// TIA Portal V15 export
// export: Created 2018-05-29T12:25:38.1552518Z, ExportSetting WithDefaults, DisplayName Totally Integrated Automation Portal, DisplayVersion V15, DisplayName STEP 7 Professional, DisplayVersion V15, DisplayName WinCC Professional, DisplayVersion V15, DisplayName TIA Portal Openness, DisplayVersion V15
FUNCTION_BLOCK "phase_example"   // FB1, STL
TITLE = phase_example_fc
{ S7_Optimized_Access := 'TRUE' }
VERSION : 0.1
// phase_example
// This some general description in a comment table.
// This is a new line in the description.
// This is another comment table without borders.
// This is a new line in the 2nd table
// stored: AutoNumber true, UDAEnableTagReadback false
   VAR_INPUT
      scantime : Real;   // the scantime of this EM/phase, used to increase timers
      Bool1 : BOOL;   // - undefined
      Bool2 : BOOL;   // - undefined
      EM_I_OUT_ID : INT;   // - undefined
      Some_Dyn_EM_ID : INT;   // - undefined
      DB_NO : INT;   // - undefined
      XV003_OPN : BOOL;   // - undefined
      XV003_CLS : BOOL;   // - undefined
      XV003_MERR : BOOL;   // - undefined
      XV004_OPN : BOOL;   // - undefined
      XV004_CLS : BOOL;   // - undefined
      XV004_MERR : BOOL;   // - undefined
      XV005_OPN : BOOL;   // - undefined
      XV005_CLS : BOOL;   // - undefined
      XV005_MERR : BOOL;   // - undefined
      P001_RUN : BOOL;   // test a CM - undefined
      P001_STOP : BOOL;   // test a CM - undefined
      P001_MERR : BOOL;   // test a CM - undefined
      P001_MPS : BOOL;   // test a CM - Motor Protecting Switch
      P002_RUN : BOOL;   // test a CM where the casing doesn't match an existing type - undefined
      P002_STOP : BOOL;   // test a CM where the casing doesn't match an existing type - undefined
      P002_MERR : BOOL;   // test a CM where the casing doesn't match an existing type - undefined
      P002_MPS : BOOL;   // test a CM where the casing doesn't match an existing type - Motor Protecting Switch
      EM_I_OUT_OWN : INT;   // - undefined
      EM_I_OUT_STA : INT;   // - undefined
      EM_I_OUT_ERR : BOOL;   // - undefined
      EM_I_OUT_ERRNO : DINT;   // - undefined
      EM_I_OUT_ACTIV : BOOL;   // - undefined
      EM_I_OUT_LT : REAL;   // - undefined
      EM_I_OUT_PT : REAL;   // - undefined
      LT001_PV : REAL;   // - undefined
      LT001_AHH : BOOL;   // - undefined
      LT001_AH : BOOL;   // - undefined
      LT001_AL : BOOL;   // - undefined
      LT001_ALL : BOOL;   // - undefined
      LT001_ERR : BOOL;   // - undefined
      LT002_PV : REAL;   // - undefined
      LT002_AHH : BOOL;   // - undefined
      LT002_AH : BOOL;   // - undefined
      LT002_AL : BOOL;   // - undefined
      LT002_ALL : BOOL;   // - undefined
      LT002_ERR : BOOL;   // - undefined
      FIC001_PV : REAL;   // - undefined
      FIC001_ERR : BOOL;   // - undefined
      Some_Dyn_EM_OWN : INT;   // An example of an EM that's dynamically linked to the phase - undefined
      Some_Dyn_EM_STA : INT;   // An example of an EM that's dynamically linked to the phase - undefined
      Some_Dyn_EM_ERR : BOOL;   // An example of an EM that's dynamically linked to the phase - undefined
      Some_Dyn_EM_ERRNO : DINT;   // An example of an EM that's dynamically linked to the phase - undefined
      Some_Dyn_EM_ACTIV : BOOL;   // An example of an EM that's dynamically linked to the phase - undefined
      Some_Dyn_EM_LT : REAL;   // An example of an EM that's dynamically linked to the phase - undefined
      Some_Dyn_EM_PT : REAL;   // An example of an EM that's dynamically linked to the phase - undefined
      XV008_OPN : BOOL;   // - undefined
      XV008_CLS : BOOL;   // - undefined
      XV008_MERR : BOOL;   // - undefined
   END_VAR
   VAR_OUTPUT
      phase_id : Int;   // unique number for every phase instance over the whole project
      state : Int;
      stepnumber : Int;   // actual stepnumber
      message : DInt;   // number of the message to be displayed
      button_1_text : DInt;   // number of the text to be displayed on the button_1_text
      button_2_text : DInt;   // number of the text to be displayed on the button_2_text
      button_3_text : DInt;   // number of the text to be displayed on the button_3_text
      button_1_visible : Bool;   // 1 = visible
      button_2_visible : Bool;   // 1 = visible
      button_3_visible : Bool;   // 1 = visible
      button_reverse : Byte;   // spare
      state_idle : Bool;
      state_running : Bool;
      state_complete : Bool;
      state_pausing : Bool;
      state_paused : Bool;
      state_holding : Bool;
      state_held : Bool;
      state_restarting : Bool;
      state_stopping : Bool;
      state_stopped : Bool;
      state_aborting : Bool;
      state_aborted : Bool;
      enable_start : Bool;   // 1 start command from hmi or other operator interface
      enable_stop : Bool;   // 2 stop command from hmi or other operator interface
      enable_hold : Bool;   // 3 hold command from hmi or other operator interface
      enable_restart : Bool;   // 4 restart command from hmi or other operator interface
      enable_abort : Bool;   // 5 abort command from hmi or other operator interface
      enable_reset : Bool;   // 6 reset command from hmi or other operator interface
      enable_pause : Bool;   // 7 pause command from hmi or other operator interface
      enable_resume : Bool;   // 8 resume command from hmi or other operator interface
      enable_auto : Bool;   // 1 = auto command from plc program
      enable_man : Bool;   // 1 = manual command from plc program
      enable_byte : Bool;
      auto : Bool;
      steptime_s : Real;   // complete steptime in seconds. same value as the other steptimes
      steptime_m : Real;   // complete steptime in minutes. same value as the other steptimes
      steptime_h : Real;   // complete steptime in hours. same value as the other steptimes
      MSG_no01 : Dint;
      MSG_no02 : Dint;
      MSG_no03 : Dint;
      MSG_no04 : Dint;
      MSG_no05 : Dint;
      MSG_no06 : Dint;
      MSG_no07 : Dint;
      MSG_no08 : Dint;
      MSG_no09 : Dint;
      MSG_no10 : Dint;
      Destination : INT;   // - undefined
      setpoint : REAL;   // - undefined
      some_bool_out : BOOL;   // - undefined
      XV003_CMD : BOOL;   // - Auto command from program
      XV004_CMD : BOOL;   // - Auto command from program
      XV005_CMD : BOOL;   // - Auto command from program
      P001_ON : BOOL;   // test a CM - Switch Motor ON
      P001_AUT : BOOL;   // test a CM - Swtich Motor to AUTO
      P002_ON : BOOL;   // test a CM where the casing doesn't match an existing type - Switch Motor ON
      P002_AUT : BOOL;   // test a CM where the casing doesn't match an existing type - Swtich Motor to AUTO
      EM_I_OUT_REQ : INT;   // - undefined
      EM_I_OUT_CMD : INT;   // - undefined
      EM_I_OUT_P_SP : REAL;   // - undefined
      FIC001_EXT : BOOL;   // - Switch to External Mode
      FIC001_SP : REAL;   // - Operator Setpoint in Internal Mode
      FIC001_AUT : BOOL;   // - Switch to Auto Mode
      FIC001_VAL_OUT : REAL;   // - Operator Output Value
      FIC001_SET_SP : BOOL;   // - undefined
      FIC001_SET_OUT : BOOL;   // - undefined
      Some_Dyn_EM_REQ : INT;   // An example of an EM that's dynamically linked to the phase - undefined
      Some_Dyn_EM_CMD : INT;   // An example of an EM that's dynamically linked to the phase - undefined
      Some_Dyn_EM_P_SP : REAL;   // An example of an EM that's dynamically linked to the phase - undefined
      timer_dosing_pause : BOOL;   // timer paused - undefined
      timer_dosing_s : REAL;   // timer in seconds - undefined
      timer_dosing_m : REAL;   // timer in minutes - undefined
      timer_dosing_h : REAL;   // timer in hours - undefined
      timer_mixing_pause : BOOL;   // timer paused - undefined
      timer_mixing_s : REAL;   // timer in seconds - undefined
      timer_mixing_m : REAL;   // timer in minutes - undefined
      timer_mixing_h : REAL;   // timer in hours - undefined
      timer_circulation_pause : BOOL;   // timer paused - undefined
      timer_circulation_s : REAL;   // timer in seconds - undefined
      timer_circulation_m : REAL;   // timer in minutes - undefined
      timer_circulation_h : REAL;   // timer in hours - undefined
      XV008_CMD : BOOL;   // - Auto command from program
   END_VAR
   VAR_IN_OUT
      plc_commands : DWord;   // combined commands from the master
      hmi_commands : DWord;   // combined commands from the HMI
      hmi_par_without_unit : Real;   // - undefined
      timesetting : Real;   // - undefined
   END_VAR
   VAR DB_SPECIFIC
      previous_stepnumber : Int;   // actual stepnumber
      start_conditions : Bool;   // start conditions 1 = all good
      hold_conditions : Bool;   // hold conditions 1 = all good
      first_scan : Bool;   // first scan of the step active
      last_scan : Bool;   // last scan of the step active
      start_cond_01 : Bool;   // 1 = OK / 0 = NOK
      start_cond_02 : Bool;   // 1 = OK / 0 = NOK
      start_cond_03 : Bool;   // 1 = OK / 0 = NOK
      start_cond_04 : Bool;   // 1 = OK / 0 = NOK
      start_cond_05 : Bool;   // 1 = OK / 0 = NOK
      start_cond_06 : Bool;   // 1 = OK / 0 = NOK
      start_cond_07 : Bool;   // 1 = OK / 0 = NOK
      start_cond_08 : Bool;   // 1 = OK / 0 = NOK
      start_cond_09 : Bool;   // 1 = OK / 0 = NOK
      start_cond_10 : Bool;   // 1 = OK / 0 = NOK
      start_cond_11 : Bool;   // 1 = OK / 0 = NOK
      start_cond_12 : Bool;   // 1 = OK / 0 = NOK
      start_cond_13 : Bool;   // 1 = OK / 0 = NOK
      start_cond_14 : Bool;   // 1 = OK / 0 = NOK
      start_cond_15 : Bool;   // 1 = OK / 0 = NOK
      start_cond_16 : Bool;   // 1 = OK / 0 = NOK
      hold_cond_01 : Bool;   // 1 = OK / 0 = NOK
      hold_cond_02 : Bool;   // 1 = OK / 0 = NOK
      hold_cond_03 : Bool;   // 1 = OK / 0 = NOK
      hold_cond_04 : Bool;   // 1 = OK / 0 = NOK
      hold_cond_05 : Bool;   // 1 = OK / 0 = NOK
      hold_cond_06 : Bool;   // 1 = OK / 0 = NOK
      hold_cond_07 : Bool;   // 1 = OK / 0 = NOK
      hold_cond_08 : Bool;   // 1 = OK / 0 = NOK
      hold_cond_09 : Bool;   // 1 = OK / 0 = NOK
      hold_cond_10 : Bool;   // 1 = OK / 0 = NOK
      hold_cond_11 : Bool;   // 1 = OK / 0 = NOK
      hold_cond_12 : Bool;   // 1 = OK / 0 = NOK
      hold_cond_13 : Bool;   // 1 = OK / 0 = NOK
      hold_cond_14 : Bool;   // 1 = OK / 0 = NOK
      hold_cond_15 : Bool;   // 1 = OK / 0 = NOK
      hold_cond_16 : Bool;   // 1 = OK / 0 = NOK
      in_steprange : Bool;   // detection of steprange for holdcondition
      Module_Error : Bool;   // Error on one of the connected modules (CM or EM)
      CM_Error_no : Dint;   // Error no of the CM in error
      EM_Error_no : Dint;   // Error no of the EM in error
      "e" : Real;   // - undefined
      f : Real;   // - undefined
      g : Real;   // - undefined
      h : Real;   // - undefined
      ii : Real;   // - undefined
      j : Real;   // - undefined
      k : Real;   // - undefined
      l : Real;   // - undefined
      mm : Real;   // - undefined
      n : Real;   // - undefined
      o : Real;   // - undefined
      pp : Real;   // - undefined
      qq : Real;   // - undefined
      rr : Real;   // - undefined
      ss : Real;   // - undefined
      tt : Real;   // - undefined
      u : Real;   // - undefined
      v : Real;   // - undefined
      ww : Real;   // - undefined
      xx : Real;   // - undefined
      y : Real;   // - undefined
      z : Real;   // - undefined
      foo : Real;   // - undefined
      bar : Real;   // - undefined
      stoplevel : Real;   // - undefined
      startlevel : Real;   // - undefined
      offset : Real;   // - undefined
      var1 : Real;   // - undefined
      test1 : Real;   // - undefined
      test2 : Real;   // - undefined
      intvar : Int;   // - undefined
      ""EM_I_OUT"" : "EM_I_OUT_UDT";   // UDT for the linked EM
      ""Some_Dyn_EM"" : "EM_I_OUT_UDT";   // UDT for the linked EM
   END_VAR
   VAR_TEMP
      plc_start : Bool;   // 1 start command from plc program
      plc_stop : Bool;   // 2 stop command from plc program
      plc_hold : Bool;   // 3 hold command from plc program
      plc_restart : Bool;   // 4 restart command from plc program
      plc_abort : Bool;   // 5 abort command from plc program
      plc_reset : Bool;   // 6 reset command from plc program
      plc_pause : Bool;   // 7 pause command from plc program
      plc_resume : Bool;   // 8 resume command from plc program
      plc_auto : Bool;   // 0 manual,1 auto command from plc program
      plc_man : Bool;   // 0 manual,1 auto command from plc program
      plc_cmd : Bool;
      hmi_start : Bool;   // 1 start command from hmi or other operator interface
      hmi_stop : Bool;   // 2 stop command from hmi or other operator interface
      hmi_hold : Bool;   // 3 hold command from hmi or other operator interface
      hmi_restart : Bool;   // 4 restart command from hmi or other operator interface
      hmi_abort : Bool;   // 5 abort command from hmi or other operator interface
      hmi_reset : Bool;   // 6 reset command from hmi or other operator interface
      hmi_pause : Bool;   // 7 pause command from hmi or other operator interface
      hmi_resume : Bool;   // 8 resume command from hmi or other operator interface
      hmi_auto : Bool;   // 1 auto command from plc program
      hmi_man : Bool;   // 0 manual command from plc program
      hmi_cmd : Bool;
      hmi_BTN1 : Bool;
      hmi_BTN2 : Bool;
      hmi_BTN3 : Bool;
      command_start : Bool;   // 1 start command from plc or hmi
      command_stop : Bool;   // 2 stop command from plc or hmi
      command_hold : Bool;   // 3 hold command from plc or hmi
      command_restart : Bool;   // 4 restart command from plc or hmi
      command_abort : Bool;   // 5 abort command from plc or hmi
      command_reset : Bool;   // 6 reset command from plc or hmi
      command_pause : Bool;   // 7 pause command from plc or hmi
      command_resume : Bool;   // 8 resume command from plc or hmi
      command_auto : Bool;   // 1 auto command from plc or hmi
      command_man : Bool;   // 0 auto command from plc or hmi
      command_cmd : Bool;
      button_1_pushed : Bool;   // button pushed
      button_2_pushed : Bool;   // button pushed
      button_3_pushed : Bool;   // button pushed
      sh_cond_01 : Bool;   // 1 = OK / 0 = NOK: intermediate value
      sh_cond_02 : Bool;   // 1 = OK / 0 = NOK: intermediate value
      sh_cond_03 : Bool;   // 1 = OK / 0 = NOK: intermediate value
      sh_cond_04 : Bool;   // 1 = OK / 0 = NOK: intermediate value
      sh_cond_05 : Bool;   // 1 = OK / 0 = NOK: intermediate value
      sh_cond_06 : Bool;   // 1 = OK / 0 = NOK: intermediate value
      sh_cond_07 : Bool;   // 1 = OK / 0 = NOK: intermediate value
      sh_cond_08 : Bool;   // 1 = OK / 0 = NOK: intermediate value
      sh_cond_09 : Bool;   // 1 = OK / 0 = NOK: intermediate value
      sh_cond_10 : Bool;   // 1 = OK / 0 = NOK: intermediate value
      sh_cond_11 : Bool;   // 1 = OK / 0 = NOK: intermediate value
      sh_cond_12 : Bool;   // 1 = OK / 0 = NOK: intermediate value
      sh_cond_13 : Bool;   // 1 = OK / 0 = NOK: intermediate value
      sh_cond_14 : Bool;   // 1 = OK / 0 = NOK: intermediate value
      sh_cond_15 : Bool;   // 1 = OK / 0 = NOK: intermediate value
      sh_cond_16 : Bool;   // 1 = OK / 0 = NOK: intermediate value
      initial_scan : Bool;   // pulse active on the first cycle of a new scan
      Temp_stepnumber : Int;   // actual stepnumber
      V1 : Real;   // intermediate value for calculation
      V2 : Real;   // intermediate value for calculation
      V3 : Real;   // intermediate value for calculation
      V4 : Real;   // intermediate value for calculation
      V5 : Real;   // intermediate value for calculation
      V6 : Real;   // intermediate value for calculation
      V7 : Real;   // intermediate value for calculation
      V8 : Real;   // intermediate value for calculation
      V9 : Real;   // intermediate value for calculation
      V10 : Real;   // intermediate value for calculation
      V11 : Real;   // intermediate value for calculation
      V12 : Real;   // intermediate value for calculation
      V13 : Real;   // intermediate value for calculation
      V14 : Real;   // intermediate value for calculation
      V15 : Real;   // intermediate value for calculation
      V16 : Real;   // intermediate value for calculation
      V17 : Real;   // intermediate value for calculation
      B1 : Real;   // intermediate value for calculation
      B2 : Real;   // intermediate value for calculation
      B3 : Real;   // intermediate value for calculation
      B4 : Real;   // intermediate value for calculation
      B5 : Real;   // intermediate value for calculation
      B6 : Real;   // intermediate value for calculation
      B7 : Real;   // intermediate value for calculation
      B8 : Real;   // intermediate value for calculation
      B9 : Real;   // intermediate value for calculation
      B10 : Real;   // intermediate value for calculation
      B11 : Real;   // intermediate value for calculation
      B12 : Real;   // intermediate value for calculation
      B13 : Real;   // intermediate value for calculation
      B14 : Real;   // intermediate value for calculation
      B15 : Real;   // intermediate value for calculation
      B16 : Real;   // intermediate value for calculation
      B17 : Real;   // intermediate value for calculation
   END_VAR
BEGIN

NETWORK
TITLE = INDEX
// ___phase_example_Step_0_
// ___phase_example_Step_10_
// ___phase_example_Step_20_
// ___phase_example_Step_30_
// ___phase_example_Step_40_
// ___phase_example_Step_50_
// ___phase_example_Step_70_
// ___phase_example_Step_80_
// ___phase_example_Step_90_
// ___phase_example_Step_100_
// ___phase_example_Step_120_
// ___phase_example_Step_130_
// ___phase_example_Step_150_
// ___phase_example_Step_170_
// ___phase_example_Step_180_
// ___phase_example_Step_190_
// ___phase_example_Step_200_
// ___phase_example_Step_230_
// ___phase_example_Step_250_
// ___phase_example_Step_260_
// ___phase_example_Step_280_
// ___phase_example_Step_300_
// ___phase_example_Step_310_
// ___phase_example_Step_320_
// ___phase_example_Step_330_
// ___phase_example_Step_340_
// ___phase_example_Step_350_
// ___phase_example_Step_360_
// ___phase_example_Step_370_
// ___phase_example_Step_420_
// ___phase_example_Step_430_
// ___phase_example_Step_440_
// ___phase_example_Step_450_
// ___phase_example_Step_460_
// ___phase_example_Step_470_
// ___phase_example_Step_480_
// ___phase_example_Step_490_
// ___phase_example_Step_510_
// ___phase_example_Step_520_
// ___phase_example_Step_530_
// ___phase_example_Step_540_
// ___phase_example_Step_550_
// ___phase_example_Step_560_
// ___phase_example_Step_570_
// ___phase_example_Step_580_
// ___phase_example_Step_590_
// ___phase_example_Step_600_
// ___phase_example_Step_610_
// ___phase_example_Step_640_
// ___phase_example_Step_650_
// ___phase_example_Step_660_
// ___phase_example_Step_670_
// ___phase_example_Step_680_
// ___phase_example_Step_690_
// ___phase_example_Step_700_
// ___phase_example_Step_710_
// ___phase_example_Step_720_
// ___phase_example_Step_730_
// ___phase_example_Step_740_
// ___phase_example_Step_750_
// ___phase_example_Step_760_
// ___phase_example_Step_770_
// ___phase_example_Step_780_
// ___phase_example_Step_790_
// ___phase_example_Step_810_
// ___phase_example_Step_820_
// ___phase_example_Step_830_
// ___phase_example_Step_840_
// ___phase_example_Step_850_
// ___phase_example_Step_860_
// ___phase_example_Step_870_
// ___phase_example_Step_880_
// ___phase_example_Step_890_
// ___phase_example_Step_910_
// ___phase_example_Step_920_
// ___phase_example_Step_930_
// ___phase_example_Step_940_
// ___phase_example_Step_950_
// ___phase_example_Step_960_
// ___phase_example_Step_970_
// ___phase_example_Step_980_
// ___phase_example_Step_990_
// ___phase_example_Step_1000_
// ___phase_example_Step_8000_
// empty



NETWORK
TITLE = Phase ID
// Make the Phase ID based on its DB number
      L     DINO;
      T     #phase_id;



NETWORK
TITLE = Read EMs
// network comment


      CALL  "em_read"
      ( EM_ID               := "EM_I_OUT_ID",
        UDT_LOCATION        := #EM_I_OUT,
        UDT_OFFSET          := #"40",
        Length              := #"40",
        EM_addressing_error := #"M      0.0"
      );

      CALL  "em_read"
      ( EM_ID               := "Some_Dyn_EM_ID",
        UDT_LOCATION        := #Some_Dyn_EM,
        UDT_OFFSET          := #"40",
        Length              := #"40",
        EM_addressing_error := #"M      0.0"
      );



NETWORK
TITLE = HMI Commands
// Get the commands from the HMI that have been received in the last cycle
// They come in a DWORD to save tags
// They need to be transferred to BOOLS for easy use
// Once transferred then clear the DWORD so new commands can be detected in the next cycle
// Load the command from the HMI in AR1
      LAR1  P##hmi_commands;  //Command from WinCC

// copy all commands to the bools

      A     DBB [AR1, P#3.0];  //WinCC tag bit 0
      =     #hmi_start;

      A     DBB [AR1, P#3.1];  //WinCC tag bit 1
      =     #hmi_stop;

      A     DBB [AR1, P#3.2];  //WinCC tag bit 2
      =     #hmi_hold;

      A     DBB [AR1, P#3.3];  //WinCC tag bit 3
      =     #hmi_restart;

      A     DBB [AR1, P#3.4];  //WinCC tag bit 4
      =     #hmi_abort;

      A     DBB [AR1, P#3.5];  //WinCC tag bit 5
      =     #hmi_reset;

      A     DBB [AR1, P#3.6];  //WinCC tag bit 6
      =     #hmi_pause;

      A     DBB [AR1, P#3.7];  //WinCC tag bit 7
      =     #hmi_resume;

      A     DBB [AR1, P#2.0];  //WinCC tag bit 8
      =     #hmi_auto;

      A     DBB [AR1, P#2.1];  //WinCC tag bit 9
      =     #hmi_man;

      A     DBB [AR1, P#2.2];  //WinCC tag bit 10
      =     #hmi_BTN1;

      A     DBB [AR1, P#2.3];  //WinCC tag bit 11
      =     #hmi_BTN2;

      A     DBB [AR1, P#2.4];  //WinCC tag bit 12
      =     #hmi_BTN3;



NETWORK
TITLE = plc Commands
// Get the commands from the HMI that have been received in the last cycle
// They come in a DWORD to save tags
// They need to be transferred to BOOLS for easy use
// Once transferred then clear the DWORD so new commands can be detected in the next cycle
      LAR1  P##plc_commands;  //Command from program

// copy all commands to the bools

      A     DBB [AR1, P#3.0];  //WinCC tag bit 0
      =     #plc_start;

      A     DBB [AR1, P#3.1];  //WinCC tag bit 1
      =     #plc_stop;

      A     DBB [AR1, P#3.2];  //WinCC tag bit 2
      =     #plc_hold;

      A     DBB [AR1, P#3.3];  //WinCC tag bit 3
      =     #plc_restart;

      A     DBB [AR1, P#3.4];  //WinCC tag bit 4
      =     #plc_abort;

      A     DBB [AR1, P#3.5];  //WinCC tag bit 5
      =     #plc_reset;

      A     DBB [AR1, P#3.6];  //WinCC tag bit 6
      =     #plc_pause;

      A     DBB [AR1, P#3.7];  //WinCC tag bit 7
      =     #plc_resume;

      A     DBB [AR1, P#2.0];  //WinCC tag bit 8
      =     #plc_auto;

      A     DBB [AR1, P#2.1];  //WinCC tag bit 9
      =     #plc_man;

//A     DIX [AR1,P#2.2] 	// WinCC tag bit 10
//= plc_BTN1

//A     DIX [AR1,P#2.3] 	// WinCC tag bit 11
//= plc_start

//A     DIX [AR1,P#2.4] 	// WinCC tag bit 12
//= plc_start


// reset operator command
      L     DW#16#F000;
      T     #hmi_commands;
      T     #plc_commands;



NETWORK
TITLE = Combined Commands
// Combine the commands from the HMI and PLC in one command
// (OR-function)
      O     #plc_start;
      O     #hmi_start;
      =     #command_start;

      O     #plc_stop;
      O     #hmi_stop;
      =     #command_stop;

      O     #plc_hold;
      O     #hmi_hold;
      =     #command_hold;

      O     #plc_restart;
      O     #hmi_restart;
      =     #command_restart;

      O     #plc_abort;
      O     #hmi_abort;
      =     #command_abort;

      O     #plc_reset;
      O     #hmi_reset;
      =     #command_reset;

      O     #plc_pause;
      O     #hmi_pause;
      =     #command_pause;

      O     #plc_resume;
      O     #hmi_resume;
      =     #command_resume;

      O     #plc_auto;
      O     #hmi_auto;
      =     #command_auto;

      O     #plc_man;
      O     #hmi_man;
      =     #command_man;

      A     #command_auto;
      S     #auto;

      A     #command_man;
      R     #auto;

      CLR;
      =     #enable_man;
      =     #enable_auto;

      A     #auto;
      =     #enable_man;

      AN    #auto;
      =     #enable_auto;


      A     #hmi_BTN1;
      =     #button_1_pushed;

      A     #hmi_BTN2;
      =     #button_2_pushed;

      A     #hmi_BTN3;
      =     #button_3_pushed;



NETWORK
TITLE = Steptimers
// If the previous stepnumber is not the same as the current one
// then reset the timers, else increase them
// This is at the start of the FB because normal stepchanges will take
// till the next cycle to become active
// check if stepnumber == previous_stepnumber
      L     #stepnumber;
      L     #previous_stepnumber;
      ==I;  //if condition true then {
      JCN   TIM1;

// increase timer
      L     #scantime;
      L     #steptime_s;
      +R;
      T     #steptime_s;

      JU    TIM2;
TIM1: NOP   0;

// reset timer
      L     0.0;
      T     #steptime_s;

TIM2: NOP   0;  //end if

// calculate the other two timers
      L     #steptime_s;
      L     60.0;
      /R;
      T     #steptime_m;

      L     60.0;
      /R;
      T     #steptime_h;



NETWORK
TITLE = Other Timers
// If timers are needed that cannot be solved with the steptime.
// Timers need to start with the name 'timer'
// They are paused by default
// They can be unpaused
// They can be reset by writing the value to 0 in the action
// Every timer is available in s, m and h


//--------------------------------
// timer_dosing
//
//--------------------------------

      AN    #timer_dosing_pause;  //if not paused ...
      JCN   TI1;

      L     #scantime;  //increase the timer
      L     #timer_dosing_s;
      +R;
      T     #timer_dosing_s;

TI1:  NOP   0;  //end if

// calculate the other two timers
      L     #timer_dosing_s;
      L     60.0;
      /R;
      T     #timer_dosing_m;

      L     60.0;
      /R;
      T     #timer_dosing_h;

//--------------------------------
// timer_mixing
//
//--------------------------------

      AN    #timer_mixing_pause;  //if not paused ...
      JCN   TI2;

      L     #scantime;  //increase the timer
      L     #timer_mixing_s;
      +R;
      T     #timer_mixing_s;

TI2:  NOP   0;  //end if

// calculate the other two timers
      L     #timer_mixing_s;
      L     60.0;
      /R;
      T     #timer_mixing_m;

      L     60.0;
      /R;
      T     #timer_mixing_h;

//--------------------------------
// timer_circulation
//
//--------------------------------

      AN    #timer_circulation_pause;  //if not paused ...
      JCN   TI3;

      L     #scantime;  //increase the timer
      L     #timer_circulation_s;
      +R;
      T     #timer_circulation_s;

TI3:  NOP   0;  //end if

// calculate the other two timers
      L     #timer_circulation_s;
      L     60.0;
      /R;
      T     #timer_circulation_m;

      L     60.0;
      /R;
      T     #timer_circulation_h;



NETWORK
TITLE = detect initial scan
// create a pulse active on the first cycle of a new scan
// this signal can be used in the step to execute some actions in the first cycle of the step
      L     #stepnumber;
      L     #previous_stepnumber;
      <>I;
      =     #initial_scan;



NETWORK
TITLE = Save old step
// Save old step
      L     #stepnumber;
      T     #previous_stepnumber;



NETWORK
TITLE = Change States
// Change States
// --------------------------------
// This phase template is design to let the stepnumber be the single
// source of truth for the state of the phase.
// All other indicators of state from this phase are deducted from the
// stepnumber.
// And the state can only be changed by changing the stepnumber 
// For every state we both create a bit, and an integer value
// Both have the same meaning and can be chosen for usage based
// on what is most convenient
//--------------------------------
// Stop Command
//--------------------------------

      A     #enable_stop;
      A     #command_stop;  //stop command

      JCN   CM02;

      L     0;  //config: target step for this command (-1 if not used)
      T     #stepnumber;

CM02: NOP   0;

//--------------------------------
// Hold Command
//--------------------------------

      A     #enable_hold;
      A(;
      O     #command_hold;  //hold command
      ON    #hold_conditions;  //hold condition active, configured outside this FB
      );
      JCN   CM03;

      L     8000;  //config: target step for this command (-1 if not used)
      T     #stepnumber;

CM03: NOP   0;

//--------------------------------
// Abort Command
//--------------------------------

      A     #enable_abort;
      A     #command_abort;  //abort command
      JCN   CM05;

// Disabled in this config because we only want to allow abort when held
      L     9000;  //config: target step for this command (-1 if not used)
      T     #stepnumber;

CM05: NOP   0;

//--------------------------------
// Pause Command
//--------------------------------

      A     #enable_pause;
      A     #command_pause;  //pause command
      JCN   CM06;

      L     6000;  //config: target step for this command (-1 if not used)
      T     #stepnumber;

CM06: NOP   0;



NETWORK
TITLE = Phase States
// Update Phase States based on the stepnumber
// 0 idle 
// 1 running
// 2 completed
// 3 pausing
// 4 paused
// 5 holding
// 6 held
// 7 restarting
// 8 stopping
// 9 stopped
// 10 aborting
// 11 aborted
// -------------------------------
// See previous network for explanation
//--------------------------------
// Disable all permissions for the commands
// The individial permissions will be set again
// in the next steps depending on the state
//--------------------------------

      CLR;
      =     #enable_start;
      =     #enable_stop;
      =     #enable_hold;
      =     #enable_restart;
//	=	enable_abort
      =     #enable_reset;
      =     #enable_pause;
      =     #enable_resume;

//--------------------------------
// 0 Idle state based on stepnumber
//--------------------------------
      L     0;  //config: lowest step (-1 if state not used)
      L     #stepnumber;
      >=I;
      L     0;  //config: highest step (-1 if state not used)
      <=I;
      =     #state_idle;  //update state bit
      JCN   ST00;

// update state as integer
      L     0;
      T     #state;

// enable commands
      SET;
      =     #enable_start;

ST00: NOP   0;

//--------------------------------
// 1 Running state based on stepnumber
//--------------------------------
      L     1;  //config: lowest step (-1 if state not used)
      L     #stepnumber;
      <=I;
      L     9999;  //config: highest step (-1 if state not used)
      <=I;
      =     #state_running;  //update state bit
      JCN   ST01;

// update state as integer
      L     1;
      T     #state;

// enable commands
      SET;
      =     #enable_stop;
      =     #enable_hold;
//	=	enable_abort
      =     #enable_pause;

ST01: NOP   0;

//--------------------------------
// 2 Completed state based on stepnumber
//--------------------------------
      L     700;  //config: lowest step (-1 if state not used)
      L     #stepnumber;
      <=I;
      L     1000;  //config: highest step (-1 if state not used)
      <=I;
      =     #state_complete;  //update state bit
      JCN   ST02;

// update state as integer
      L     2;
      T     #state;

// enable commands
      SET;
      =     #enable_reset;

ST02: NOP   0;

//--------------------------------
// 3 Pausing state based on stepnumber
//--------------------------------
      L     6000;  //config: lowest step (-1 if state not used)
      L     #stepnumber;
      <=I;
      L     6900;  //config: highest step (-1 if state not used)
      <I;
      =     #state_pausing;  //update state bit
      JCN   ST03;

// update state as integer
      L     3;
      T     #state;

// enable commands
      SET;
      =     #enable_stop;
      =     #enable_hold;
//	=	enable_abort


ST03: NOP   0;

//--------------------------------
// 4 Paused state based on stepnumber
//--------------------------------
      L     6900;  //config: lowest step (-1 if state not used)
      L     #stepnumber;
      <=I;
      L     6999;  //config: highest step (-1 if state not used)
      <=I;
      =     #state_paused;  //update state bit
      JCN   ST04;

// update state as integer
      L     4;
      T     #state;

// enable commands
      SET;
      =     #enable_stop;
      =     #enable_hold;
//	=	enable_abort
      =     #enable_resume;

ST04: NOP   0;

//--------------------------------
// 5 Holding state based on stepnumber
//--------------------------------
      L     8000;  //config: lowest step (-1 if state not used)
      L     #stepnumber;
      <=I;
      L     8900;  //config: highest step (-1 if state not used)
      <I;
      =     #state_holding;  //update state bit
      JCN   ST05;

// update state as integer
      L     5;
      T     #state;

// enable commands
      SET;
      =     #enable_stop;
//	=	enable_abort

ST05: NOP   0;

//--------------------------------
// 6 Held state based on stepnumber
//--------------------------------
      L     8900;  //config: lowest step (-1 if state not used)
      L     #stepnumber;
      <=I;
      L     8999;  //config: highest step (-1 if state not used)
      <=I;
      =     #state_held;  //update state bit
      JCN   ST06;

// update state as integer
      L     6;
      T     #state;

// enable commands
      SET;
      =     #enable_stop;
      =     #enable_restart;
      =     #enable_abort;

ST06: NOP   0;

//--------------------------------
// 7 Restarting state based on stepnumber
//--------------------------------
      L     5000;  //config: lowest step (-1 if state not used)
      L     #stepnumber;
      <=I;
      L     5900;  //config: highest step (-1 if state not used)
      <=I;
      =     #state_restarting;  //update state bit
      JCN   ST07;

// update state as integer
      L     7;
      T     #state;

// enable commands
      SET;
      =     #enable_stop;
      =     #enable_hold;
//	=	enable_abort

ST07: NOP   0;

//--------------------------------
// 8 Stopping state based on stepnumber
//--------------------------------
      L     7000;  //config: lowest step (-1 if state not used)
      L     #stepnumber;
      <=I;
      L     7900;  //config: highest step (-1 if state not used)
      <I;
      =     #state_stopping;  //update state bit
      JCN   ST08;

// update state as integer
      L     8;
      T     #state;

// enable commands
      SET;
//	=	enable_abort

ST08: NOP   0;

//--------------------------------
// 9 Stopped state based on stepnumber
//--------------------------------
      L     7900;  //config: lowest step (-1 if state not used)
      L     #stepnumber;
      <=I;
      L     7999;  //config: highest step (-1 if state not used)
      <=I;
      =     #state_stopped;  //update state bit
      JCN   ST09;

// update state as integer
      L     9;
      T     #state;

// enable commands
      SET;
//	=	enable_abort
      =     #enable_reset;

ST09: NOP   0;

//--------------------------------
// 10 Aborting state based on stepnumber
//--------------------------------
      L     9000;  //config: lowest step (-1 if state not used)
      L     #stepnumber;
      <=I;
      L     9900;  //config: highest step (-1 if state not used)
      <I;
      =     #state_aborting;  //update state bit
      JCN   ST10;

// update state as integer
      L     10;
      T     #state;

ST10: NOP   0;

//--------------------------------
// 11 Aborted state based on stepnumber
//--------------------------------
      L     9900;  //config: lowest step (-1 if state not used)
      L     #stepnumber;
      <=I;
      L     9999;  //config: highest step (-1 if state not used)
      <=I;
      =     #state_aborted;  //update state bit
      JCN   ST11;

// update state as integer
      L     11;
      T     #state;

// enable commands
      SET;
      =     #enable_reset;

ST11: NOP   0;


//--------------------------------
// Disable start command anyway if the start_conditions are not ok
//--------------------------------

      AN    #start_conditions;
      R     #enable_start;




NETWORK
TITLE = Collect the errors from the connected Modules (CMs and EMs)
// network comment
      CLR;
      O     #XV003_MERR;
      O     #XV004_MERR;
      O     #XV005_MERR;
      O     #P001_MERR;
      O     #P001_MPS;
      O     #P002_MERR;
      O     #P002_MPS;
      O     "EM_I_OUT".CM_error;
      O     #LT001_ERR;
      O     #LT002_ERR;
      O     #FIC001_ERR;
      O     "Some_Dyn_EM".CM_error;
      O     #XV008_MERR;
      =     #Module_Error;



NETWORK
TITLE = Assign a message number to each error
// This code tries to assign an error message to each CM error
// If multiple CMs have an error then it only stores one
// This is the phase type so we don't know which CM/EM instance is connected
// So the error only contains the general name of the CM/EM instance
// If the actual name needs to be shown then it could be deducted
// at a higher level using the CM/EM name and phase instance
      CLR;

// clear the error no
      L     0;
      T     #CM_Error_no;
      T     #EM_Error_no;



      A     #XV003_MERR;
      JCN   E1;

      L     57;  //'CM error: XV003_MERR'
      T     #CM_Error_no;

E1:   NOP   0;

      A     #XV004_MERR;
      JCN   E2;

      L     58;  //'CM error: XV004_MERR'
      T     #CM_Error_no;

E2:   NOP   0;

      A     #XV005_MERR;
      JCN   E3;

      L     59;  //'CM error: XV005_MERR'
      T     #CM_Error_no;

E3:   NOP   0;

      A     #P001_MERR;
      JCN   E4;

      L     60;  //'CM error: P001_MERR'
      T     #CM_Error_no;

E4:   NOP   0;

      A     #P001_MPS;
      JCN   E5;

      L     61;  //'CM error: P001_MPS'
      T     #CM_Error_no;

E5:   NOP   0;

      A     #P002_MERR;
      JCN   E6;

      L     62;  //'CM error: P002_MERR'
      T     #CM_Error_no;

E6:   NOP   0;

      A     #P002_MPS;
      JCN   E7;

      L     63;  //'CM error: P002_MPS'
      T     #CM_Error_no;

E7:   NOP   0;

      A     "EM_I_OUT".CM_error;
      JCN   E8;

      L     "EM_I_OUT".CM_error_no;
      T     #CM_Error_no;

      L     64;  //'EM error: EM_I_OUT_ERR'
      T     #EM_Error_no;

E8:   NOP   0;

      A     #LT001_ERR;
      JCN   E9;

      L     65;  //'CM error: LT001_ERR'
      T     #CM_Error_no;

E9:   NOP   0;

      A     #LT002_ERR;
      JCN   E10;

      L     66;  //'CM error: LT002_ERR'
      T     #CM_Error_no;

E10:  NOP   0;

      A     #FIC001_ERR;
      JCN   E11;

      L     67;  //'CM error: FIC001_ERR'
      T     #CM_Error_no;

E11:  NOP   0;

      A     "Some_Dyn_EM".CM_error;
      JCN   E12;

      L     "Some_Dyn_EM".CM_error_no;
      T     #CM_Error_no;

      L     68;  //'EM error: Some_Dyn_EM_ERR'
      T     #EM_Error_no;

E12:  NOP   0;

      A     #XV008_MERR;
      JCN   E13;

      L     69;  //'CM error: XV008_MERR'
      T     #CM_Error_no;

E13:  NOP   0;



NETWORK
TITLE = Start and Hold Conditions
// network comment
      SET;
      =     #start_conditions;
      =     #hold_conditions;  //true = safe condition



NETWORK
TITLE = START OF THE STEPS AND TRANSITIONS
// ################################
// ################################
// Placeholder network to indicate the start of the actual sequence
// ################################	  
// ################################
// empty placeholder network



NETWORK
TITLE = Step 0
// Test step with only a comment and transition
// skip this network if stepnumber not equal to 0
      L     #stepnumber;
      L     0;
      ==I;
      JCN   J1;

//---------------------------------
// Actions (continuouss)
//---------------------------------

//---------------------------------
// --- TRANSITION TO S10 ---
//---------------------------------

// Transition Logic
      SET;  //make sure RLO is high so the transition can happen when no conditions present

      JCN   L1;

      L     10;
      T     #stepnumber;

L1:   NOP   0;


D1:   NOP   0;

//---------------------------------
// End of network: jump here if step not active
// Jump to end of this FB if the step has been active to avoid
// execution of another step in the same scan
//---------------------------------
      JU    ENDS;
J1:   NOP   0;



NETWORK
TITLE = Step 10
// Test multiple comments
// this is another line
// skip this network if stepnumber not equal to 10
      L     #stepnumber;
      L     10;
      ==I;
      JCN   J2;

//---------------------------------
// Actions (continuouss)
//---------------------------------

//---------------------------------
// --- TRANSITION TO S20 ---
//---------------------------------

// Transition Logic
      SET;  //make sure RLO is high so the transition can happen when no conditions present

      JCN   L2;

      L     20;
      T     #stepnumber;

L2:   NOP   0;


D2:   NOP   0;

//---------------------------------
// End of network: jump here if step not active
// Jump to end of this FB if the step has been active to avoid
// execution of another step in the same scan
//---------------------------------
      JU    ENDS;
J2:   NOP   0;



NETWORK
TITLE = Step 20
// Test some spacing before the comment
// Test some spacing before the first comment word
// skip this network if stepnumber not equal to 20
      L     #stepnumber;
      L     20;
      ==I;
      JCN   J3;

//---------------------------------
// Actions (continuouss)
//---------------------------------

//---------------------------------
// --- TRANSITION TO S30 ---
//---------------------------------

// Transition Logic
      SET;  //make sure RLO is high so the transition can happen when no conditions present

      JCN   L3;

      L     30;
      T     #stepnumber;

L3:   NOP   0;


D3:   NOP   0;

//---------------------------------
// End of network: jump here if step not active
// Jump to end of this FB if the step has been active to avoid
// execution of another step in the same scan
//---------------------------------
      JU    ENDS;
J3:   NOP   0;



NETWORK
TITLE = Step 30
// test a simple assignment with a variable
// skip this network if stepnumber not equal to 30
      L     #stepnumber;
      L     30;
      ==I;
      JCN   J4;

//---------------------------------
// Actions (continuouss)
//---------------------------------

// Action: e = f
      L     #f;
      T     #"e";

//---------------------------------
// --- TRANSITION TO S40 ---
//---------------------------------

// Transition Logic
      SET;  //make sure RLO is high so the transition can happen when no conditions present

      JCN   L4;

      L     40;
      T     #stepnumber;

L4:   NOP   0;


D4:   NOP   0;

//---------------------------------
// End of network: jump here if step not active
// Jump to end of this FB if the step has been active to avoid
// execution of another step in the same scan
//---------------------------------
      JU    ENDS;
J4:   NOP   0;



NETWORK
TITLE = Step 40
// test a simple assignment with a REAL
// skip this network if stepnumber not equal to 40
      L     #stepnumber;
      L     40;
      ==I;
      JCN   J5;

//---------------------------------
// Actions (continuouss)
//---------------------------------

// Action: setpoint = 25.0
      L     25.0;
      T     #setpoint;

//---------------------------------
// --- TRANSITION TO S50 ---
//---------------------------------

// Transition Logic
      SET;  //make sure RLO is high so the transition can happen when no conditions present

      JCN   L5;

      L     50;
      T     #stepnumber;

L5:   NOP   0;


D5:   NOP   0;

//---------------------------------
// End of network: jump here if step not active
// Jump to end of this FB if the step has been active to avoid
// execution of another step in the same scan
//---------------------------------
      JU    ENDS;
J5:   NOP   0;



NETWORK
TITLE = Step 50
// test a simple assignment with some BOOLS
// skip this network if stepnumber not equal to 50
      L     #stepnumber;
      L     50;
      ==I;
      JCN   J6;

//---------------------------------
// Actions (continuouss)
//---------------------------------

// Action: XV003_CMD = true
      SET;
      =     #XV003_CMD;

// Action: XV004_CMD = false
      CLR;
      =     #XV004_CMD;

//---------------------------------
// --- TRANSITION TO S70 ---
//---------------------------------

// Transition Logic
      SET;  //make sure RLO is high so the transition can happen when no conditions present

      JCN   L6;

      L     70;
      T     #stepnumber;

L6:   NOP   0;


D6:   NOP   0;

//---------------------------------
// End of network: jump here if step not active
// Jump to end of this FB if the step has been active to avoid
// execution of another step in the same scan
//---------------------------------
      JU    ENDS;
J6:   NOP   0;



NETWORK
TITLE = Step 70
// test opening a valve
// skip this network if stepnumber not equal to 70
      L     #stepnumber;
      L     70;
      ==I;
      JCN   J7;

//---------------------------------
// Actions (continuouss)
//---------------------------------

// Action: open XV003
      SET;
      =     #XV003_CMD;

//---------------------------------
// --- TRANSITION TO S80 ---
//---------------------------------

// Transition Logic
      SET;  //make sure RLO is high so the transition can happen when no conditions present

      JCN   L7;

      L     80;
      T     #stepnumber;

L7:   NOP   0;


D7:   NOP   0;

//---------------------------------
// End of network: jump here if step not active
// Jump to end of this FB if the step has been active to avoid
// execution of another step in the same scan
//---------------------------------
      JU    ENDS;
J7:   NOP   0;



NETWORK
TITLE = Step 80
// test closing a valve
// skip this network if stepnumber not equal to 80
      L     #stepnumber;
      L     80;
      ==I;
      JCN   J8;

//---------------------------------
// Actions (continuouss)
//---------------------------------

// Action: close XV003
      CLR;
      =     #XV003_CMD;

//---------------------------------
// --- TRANSITION TO S90 ---
//---------------------------------

// Transition Logic
      SET;  //make sure RLO is high so the transition can happen when no conditions present

      JCN   L8;

      L     90;
      T     #stepnumber;

L8:   NOP   0;


D8:   NOP   0;

//---------------------------------
// End of network: jump here if step not active
// Jump to end of this FB if the step has been active to avoid
// execution of another step in the same scan
//---------------------------------
      JU    ENDS;
J8:   NOP   0;



NETWORK
TITLE = Step 90
// test starting a motor
// skip this network if stepnumber not equal to 90
      L     #stepnumber;
      L     90;
      ==I;
      JCN   J9;

//---------------------------------
// Actions (continuouss)
//---------------------------------

// Action: start P001
      SET;
      =     #P001_ON;

//---------------------------------
// --- TRANSITION TO S100 ---
//---------------------------------

// Transition Logic
      SET;  //make sure RLO is high so the transition can happen when no conditions present

      JCN   L9;

      L     100;
      T     #stepnumber;

L9:   NOP   0;


D9:   NOP   0;

//---------------------------------
// End of network: jump here if step not active
// Jump to end of this FB if the step has been active to avoid
// execution of another step in the same scan
//---------------------------------
      JU    ENDS;
J9:   NOP   0;



NETWORK
TITLE = Step 100
// test stopping a motor
// skip this network if stepnumber not equal to 100
      L     #stepnumber;
      L     100;
      ==I;
      JCN   J10;

//---------------------------------
// Actions (continuouss)
//---------------------------------

// Action: stop P001
      CLR;
      =     #P001_ON;

//---------------------------------
// --- TRANSITION TO S120 ---
//---------------------------------

// Transition Logic
      SET;  //make sure RLO is high so the transition can happen when no conditions present

      JCN   L10;

      L     120;
      T     #stepnumber;

L10:  NOP   0;


D10:  NOP   0;

//---------------------------------
// End of network: jump here if step not active
// Jump to end of this FB if the step has been active to avoid
// execution of another step in the same scan
//---------------------------------
      JU    ENDS;
J10:  NOP   0;



NETWORK
TITLE = Step 120
// test with some spaces and non-matching casing => should still work
// skip this network if stepnumber not equal to 120
      L     #stepnumber;
      L     120;
      ==I;
      JCN   J11;

//---------------------------------
// Actions (continuouss)
//---------------------------------

// Action: Open XV003
      SET;
      =     #XV003_CMD;

//---------------------------------
// --- TRANSITION TO S130 ---
//---------------------------------

// Transition Logic
      SET;  //make sure RLO is high so the transition can happen when no conditions present

      JCN   L11;

      L     130;
      T     #stepnumber;

L11:  NOP   0;


D11:  NOP   0;

//---------------------------------
// End of network: jump here if step not active
// Jump to end of this FB if the step has been active to avoid
// execution of another step in the same scan
//---------------------------------
      JU    ENDS;
J11:  NOP   0;



NETWORK
TITLE = Step 130
// test enumeration
// skip this network if stepnumber not equal to 130
      L     #stepnumber;
      L     130;
      ==I;
      JCN   J12;

//---------------------------------
// Actions (continuouss)
//---------------------------------

// Action: Destination = PF-I-02
      L     2;
      T     #Destination;

//---------------------------------
// --- TRANSITION TO S150 ---
//---------------------------------

// Transition Logic
      SET;  //make sure RLO is high so the transition can happen when no conditions present

      JCN   L12;

      L     150;
      T     #stepnumber;

L12:  NOP   0;


D12:  NOP   0;

//---------------------------------
// End of network: jump here if step not active
// Jump to end of this FB if the step has been active to avoid
// execution of another step in the same scan
//---------------------------------
      JU    ENDS;
J12:  NOP   0;



NETWORK
TITLE = Step 150
// test EM command
// skip this network if stepnumber not equal to 150
      L     #stepnumber;
      L     150;
      ==I;
      JCN   J13;

//---------------------------------
// Actions (continuouss)
//---------------------------------

// Action: EM_I_OUT = Pump_Fixed_Pressure
      L     2;
      T     "EM_I_OUT".Command;

//---------------------------------
// --- TRANSITION TO S170 ---
//---------------------------------

// Transition Logic
      SET;  //make sure RLO is high so the transition can happen when no conditions present

      JCN   L13;

      L     170;
      T     #stepnumber;

L13:  NOP   0;


D13:  NOP   0;

//---------------------------------
// End of network: jump here if step not active
// Jump to end of this FB if the step has been active to avoid
// execution of another step in the same scan
//---------------------------------
      JU    ENDS;
J13:  NOP   0;



NETWORK
TITLE = Step 170
// test some simple calculations
// skip this network if stepnumber not equal to 170
      L     #stepnumber;
      L     170;
      ==I;
      JCN   J14;

//---------------------------------
// Actions (continuouss)
//---------------------------------

// Action: xx = y * z
      L     #y;
      L     #z;
      *R;
      T     #xx;

// Action: rr = e / 2.0
      L     #"e";
      L     2.0;
      /R;
      T     #rr;

// Action: g = h + ii
      L     #h;
      L     #ii;
      +R;
      T     #g;

// Action: j = k – mm
      L     #k;
      L     #mm;
      -R;
      T     #j;

// Action: n = o + 3.4
      L     #o;
      L     3.4;
      +R;
      T     #n;

// Action: pp = 7.3 / qq
      L     7.3;
      L     #qq;
      /R;
      T     #pp;

//---------------------------------
// --- TRANSITION TO S180 ---
//---------------------------------

// Transition Logic
      SET;  //make sure RLO is high so the transition can happen when no conditions present

      JCN   L14;

      L     180;
      T     #stepnumber;

L14:  NOP   0;


D14:  NOP   0;

//---------------------------------
// End of network: jump here if step not active
// Jump to end of this FB if the step has been active to avoid
// execution of another step in the same scan
//---------------------------------
      JU    ENDS;
J14:  NOP   0;



NETWORK
TITLE = Step 180
// test complex calculations
// skip this network if stepnumber not equal to 180
      L     #stepnumber;
      L     180;
      ==I;
      JCN   J15;

//---------------------------------
// Actions (continuouss)
//---------------------------------

// Calculation: ss + tt
      L     #ss;
      L     #tt;
      +R;
      T     #V1;

// Calculation: (ss + tt) / u
      L     #V1;
      L     #u;
      /R;
      T     #V2;

// Calculation: ((ss + tt) / u) * v
      L     #V2;
      L     #v;
      *R;
      T     #V3;

// Calculation: ww - xx
      L     #ww;
      L     #xx;
      -R;
      T     #V4;

// Calculation: (ww - xx) + 1.34
      L     #V4;
      L     1.34;
      +R;
      T     #V5;

// Calculation: (((ss + tt) / u) * v) / ((ww - xx) + 1.34)
      L     #V3;
      L     #V5;
      /R;
      T     #V6;

// Action: rr = (ss + tt) / u * v / (ww – xx + 1.34) + 2.3
      L     #V6;
      L     2.3;
      +R;
      T     #rr;

// Action: foo = bar + 1.0
      L     #bar;
      L     1.0;
      +R;
      T     #foo;

// Calculation: startlevel + setpoint
      L     #startlevel;
      L     #setpoint;
      +R;
      T     #V7;

// Action: stoplevel = startlevel + setpoint – offset
      L     #V7;
      L     #offset;
      -R;
      T     #stoplevel;

//---------------------------------
// --- TRANSITION TO S190 ---
//---------------------------------

// Transition Logic
      SET;  //make sure RLO is high so the transition can happen when no conditions present

      JCN   L15;

      L     190;
      T     #stepnumber;

L15:  NOP   0;


D15:  NOP   0;

//---------------------------------
// End of network: jump here if step not active
// Jump to end of this FB if the step has been active to avoid
// execution of another step in the same scan
//---------------------------------
      JU    ENDS;
J15:  NOP   0;



NETWORK
TITLE = Step 190
// add two REALs
// skip this network if stepnumber not equal to 190
      L     #stepnumber;
      L     190;
      ==I;
      JCN   J16;

//---------------------------------
// Actions (continuouss)
//---------------------------------

// Action: var1 = 3.0+2.0
      L     3.0;
      L     2.0;
      +R;
      T     #var1;

//---------------------------------
// --- TRANSITION TO S200 ---
//---------------------------------

// Transition Logic
      SET;  //make sure RLO is high so the transition can happen when no conditions present

      JCN   L16;

      L     200;
      T     #stepnumber;

L16:  NOP   0;


D16:  NOP   0;

//---------------------------------
// End of network: jump here if step not active
// Jump to end of this FB if the step has been active to avoid
// execution of another step in the same scan
//---------------------------------
      JU    ENDS;
J16:  NOP   0;



NETWORK
TITLE = Step 200
// test first and last scan actions
// skip this network if stepnumber not equal to 200
      L     #stepnumber;
      L     200;
      ==I;
      JCN   J17;

//---------------------------------
// Actions (first scan)
//---------------------------------
      A     #initial_scan;
      JCN   C17;

// Action: xx = 1.0
      L     1.0;
      T     #xx;

      JU    D17;
C17:  NOP   0;


//---------------------------------
// Actions (continuouss)
//---------------------------------

// Action: y = 2.0
      L     2.0;
      T     #y;

//---------------------------------
// --- TRANSITION TO S230 ---
//---------------------------------

// Transition Logic
      SET;  //make sure RLO is high so the transition can happen when no conditions present

      JCN   L17;

      L     230;
      T     #stepnumber;

L17:  NOP   0;


//---------------------------------
// Actions (last scan)
// This is immediately executed once the stepnumber changes
//---------------------------------
      L     #stepnumber;
      L     #previous_stepnumber;
      <>I;
      JCN   D17;

// Action: z = 3.0
      L     3.0;
      T     #z;


D17:  NOP   0;

//---------------------------------
// End of network: jump here if step not active
// Jump to end of this FB if the step has been active to avoid
// execution of another step in the same scan
//---------------------------------
      JU    ENDS;
J17:  NOP   0;



NETWORK
TITLE = Step 230
// test a transition with calculation
// skip this network if stepnumber not equal to 230
      L     #stepnumber;
      L     230;
      ==I;
      JCN   J18;

//---------------------------------
// Actions (continuouss)
//---------------------------------

//---------------------------------
// --- TRANSITION TO S250 ---
//---------------------------------

// Calculation: startlevel + setpoint
      L     #startlevel;
      L     #setpoint;
      +R;
      T     #V8;

// Calculation: (startlevel + setpoint) - offset
      L     #V8;
      L     #offset;
      -R;
      T     #V9;

// Calculation: LT001_PV >= ((startlevel + setpoint) - offset)
      L     #LT001_PV;
      L     #V9;
      >=R;
      =     #B1;

// Transition Logic
      SET;  //make sure RLO is high so the transition can happen when no conditions present

      A     #B1;  //LT001 >= startlevel + setpoint – offset
      JCN   L18;

      L     250;
      T     #stepnumber;

L18:  NOP   0;


D18:  NOP   0;

//---------------------------------
// End of network: jump here if step not active
// Jump to end of this FB if the step has been active to avoid
// execution of another step in the same scan
//---------------------------------
      JU    ENDS;
J18:  NOP   0;



NETWORK
TITLE = Step 250
// test natural language transition
// skip this network if stepnumber not equal to 250
      L     #stepnumber;
      L     250;
      ==I;
      JCN   J19;

//---------------------------------
// Actions (continuouss)
//---------------------------------

//---------------------------------
// --- TRANSITION TO S260 ---
//---------------------------------

// Transition Logic
      SET;  //make sure RLO is high so the transition can happen when no conditions present

      A     #P001_RUN;  //P001 running
      JCN   L19;

      L     260;
      T     #stepnumber;

L19:  NOP   0;


D19:  NOP   0;

//---------------------------------
// End of network: jump here if step not active
// Jump to end of this FB if the step has been active to avoid
// execution of another step in the same scan
//---------------------------------
      JU    ENDS;
J19:  NOP   0;



NETWORK
TITLE = Step 260
// test enumeration
// skip this network if stepnumber not equal to 260
      L     #stepnumber;
      L     260;
      ==I;
      JCN   J20;

//---------------------------------
// Actions (continuouss)
//---------------------------------

//---------------------------------
// --- TRANSITION TO S280 ---
//---------------------------------

// Calculation:
      L     #Destination;
      L     4;
      ==I;
      =     #B2;

// Transition Logic
      SET;  //make sure RLO is high so the transition can happen when no conditions present

      A     #B2;  //Destination = PF-I-04
      JCN   L20;

      L     280;
      T     #stepnumber;

L20:  NOP   0;


D20:  NOP   0;

//---------------------------------
// End of network: jump here if step not active
// Jump to end of this FB if the step has been active to avoid
// execution of another step in the same scan
//---------------------------------
      JU    ENDS;
J20:  NOP   0;



NETWORK
TITLE = Step 280
// test enumerated status of EM
// skip this network if stepnumber not equal to 280
      L     #stepnumber;
      L     280;
      ==I;
      JCN   J21;

//---------------------------------
// Actions (continuouss)
//---------------------------------

//---------------------------------
// --- TRANSITION TO S300 ---
//---------------------------------

// Calculation:
      L     "EM_I_OUT".Status;
      L     2;
      ==I;
      =     #B3;

// Transition Logic
      SET;  //make sure RLO is high so the transition can happen when no conditions present

      A     #B3;  //EM_I_OUT = Pump_Fixed_Pressure
      JCN   L21;

      L     300;
      T     #stepnumber;

L21:  NOP   0;


D21:  NOP   0;

//---------------------------------
// End of network: jump here if step not active
// Jump to end of this FB if the step has been active to avoid
// execution of another step in the same scan
//---------------------------------
      JU    ENDS;
J21:  NOP   0;



NETWORK
TITLE = Step 300
// test if primary suffixes are detected
// skip this network if stepnumber not equal to 300
      L     #stepnumber;
      L     300;
      ==I;
      JCN   J22;

//---------------------------------
// Actions (continuouss)
//---------------------------------

//---------------------------------
// --- TRANSITION TO S310 ---
//---------------------------------

// Calculation: 2.0 * LT001_PV
      L     2.0;
      L     #LT001_PV;
      *R;
      T     #V10;

// Calculation: LT001_PV + LT001_PV
      L     #LT001_PV;
      L     #LT001_PV;
      +R;
      T     #V11;

// Calculation: (LT001_PV + LT001_PV) - LT001_PV
      L     #V11;
      L     #LT001_PV;
      -R;
      T     #V12;

// Calculation: ((LT001_PV + LT001_PV) - LT001_PV) * LT001_PV
      L     #V12;
      L     #LT001_PV;
      *R;
      T     #V13;

// Calculation: (2.0 * LT001_PV) == (((LT001_PV + LT001_PV) - LT001_PV) * LT001_PV)
      L     #V10;
      L     #V13;
      ==R;
      =     #B4;

// Transition Logic
      SET;  //make sure RLO is high so the transition can happen when no conditions present

      A     #B4;  //2.0 * LT001 = (LT001 + LT001 – LT001) * LT001
      JCN   L22;

      L     310;
      T     #stepnumber;

L22:  NOP   0;


D22:  NOP   0;

//---------------------------------
// End of network: jump here if step not active
// Jump to end of this FB if the step has been active to avoid
// execution of another step in the same scan
//---------------------------------
      JU    ENDS;
J22:  NOP   0;



NETWORK
TITLE = Step 310
// test primary suffixes in action side
// skip this network if stepnumber not equal to 310
      L     #stepnumber;
      L     310;
      ==I;
      JCN   J23;

//---------------------------------
// Actions (continuouss)
//---------------------------------

// Calculation: LT001_PV + LT001_PV
      L     #LT001_PV;
      L     #LT001_PV;
      +R;
      T     #V14;

// Calculation: (LT001_PV + LT001_PV) - LT001_PV
      L     #V14;
      L     #LT001_PV;
      -R;
      T     #V15;

// Action: test1 = (LT001 + LT001 – LT001) * LT001
      L     #V15;
      L     #LT001_PV;
      *R;
      T     #test1;

// Action: test2 = LT002
      L     #LT002_PV;
      T     #test2;

//---------------------------------
// --- TRANSITION TO S320 ---
//---------------------------------

// Transition Logic
      SET;  //make sure RLO is high so the transition can happen when no conditions present

      JCN   L23;

      L     320;
      T     #stepnumber;

L23:  NOP   0;


D23:  NOP   0;

//---------------------------------
// End of network: jump here if step not active
// Jump to end of this FB if the step has been active to avoid
// execution of another step in the same scan
//---------------------------------
      JU    ENDS;
J23:  NOP   0;



NETWORK
TITLE = Step 320
// test with AND in front
// skip this network if stepnumber not equal to 320
      L     #stepnumber;
      L     320;
      ==I;
      JCN   J24;

//---------------------------------
// Actions (continuouss)
//---------------------------------

//---------------------------------
// --- TRANSITION TO S330 ---
//---------------------------------

// Transition Logic
      SET;  //make sure RLO is high so the transition can happen when no conditions present

      A     #XV003_OPN;  //XV003 opened
      JCN   L24;

      L     330;
      T     #stepnumber;

L24:  NOP   0;


D24:  NOP   0;

//---------------------------------
// End of network: jump here if step not active
// Jump to end of this FB if the step has been active to avoid
// execution of another step in the same scan
//---------------------------------
      JU    ENDS;
J24:  NOP   0;



NETWORK
TITLE = Step 330
// test multiple conditions without explicit logic
// skip this network if stepnumber not equal to 330
      L     #stepnumber;
      L     330;
      ==I;
      JCN   J25;

//---------------------------------
// Actions (continuouss)
//---------------------------------

//---------------------------------
// --- TRANSITION TO S340 ---
//---------------------------------

// Transition Logic
      SET;  //make sure RLO is high so the transition can happen when no conditions present

      A     #XV003_OPN;  //XV003 opened
      A     #XV004_OPN;  //XV004 opened
      JCN   L25;

      L     340;
      T     #stepnumber;

L25:  NOP   0;


D25:  NOP   0;

//---------------------------------
// End of network: jump here if step not active
// Jump to end of this FB if the step has been active to avoid
// execution of another step in the same scan
//---------------------------------
      JU    ENDS;
J25:  NOP   0;



NETWORK
TITLE = Step 340
// test multiple conditions with logic
// skip this network if stepnumber not equal to 340
      L     #stepnumber;
      L     340;
      ==I;
      JCN   J26;

//---------------------------------
// Actions (continuouss)
//---------------------------------

//---------------------------------
// --- TRANSITION TO S350 ---
//---------------------------------

// Transition Logic
      SET;  //make sure RLO is high so the transition can happen when no conditions present

      A     #XV003_OPN;  //XV003 opened
      A     #XV004_OPN;  //XV004 opened
      JCN   L26;

      L     350;
      T     #stepnumber;

L26:  NOP   0;


D26:  NOP   0;

//---------------------------------
// End of network: jump here if step not active
// Jump to end of this FB if the step has been active to avoid
// execution of another step in the same scan
//---------------------------------
      JU    ENDS;
J26:  NOP   0;



NETWORK
TITLE = Step 350
// test OR-logic
// skip this network if stepnumber not equal to 350
      L     #stepnumber;
      L     350;
      ==I;
      JCN   J27;

//---------------------------------
// Actions (continuouss)
//---------------------------------

//---------------------------------
// --- TRANSITION TO S360 ---
//---------------------------------

// Transition Logic
      SET;  //make sure RLO is high so the transition can happen when no conditions present

      O     #XV003_OPN;  //XV003 opened
      O     #XV004_OPN;  //XV004 opened
      JCN   L27;

      L     360;
      T     #stepnumber;

L27:  NOP   0;


D27:  NOP   0;

//---------------------------------
// End of network: jump here if step not active
// Jump to end of this FB if the step has been active to avoid
// execution of another step in the same scan
//---------------------------------
      JU    ENDS;
J27:  NOP   0;



NETWORK
TITLE = Step 360
// test combined logic
// skip this network if stepnumber not equal to 360
      L     #stepnumber;
      L     360;
      ==I;
      JCN   J28;

//---------------------------------
// Actions (continuouss)
//---------------------------------

//---------------------------------
// --- TRANSITION TO S370 ---
//---------------------------------

// Transition Logic
      SET;  //make sure RLO is high so the transition can happen when no conditions present

      A     #XV005_OPN;  //XV005 opened
      A(;
      O     #XV003_OPN;  //XV003 opened
      O     #XV004_OPN;  //XV004 opened
      );
      JCN   L28;

      L     370;
      T     #stepnumber;

L28:  NOP   0;


D28:  NOP   0;

//---------------------------------
// End of network: jump here if step not active
// Jump to end of this FB if the step has been active to avoid
// execution of another step in the same scan
//---------------------------------
      JU    ENDS;
J28:  NOP   0;



NETWORK
TITLE = Step 370
// test improved readability
// skip this network if stepnumber not equal to 370
      L     #stepnumber;
      L     370;
      ==I;
      JCN   J29;

//---------------------------------
// Actions (continuouss)
//---------------------------------

//---------------------------------
// --- TRANSITION TO S420 ---
//---------------------------------

// Transition Logic
      SET;  //make sure RLO is high so the transition can happen when no conditions present

      A     #XV005_OPN;  //XV005 opened
      A(;
      O     #XV003_OPN;  //XV003 opened
      O     #XV004_OPN;  //XV004 opened
      );
      JCN   L29;

      L     420;
      T     #stepnumber;

L29:  NOP   0;


D29:  NOP   0;

//---------------------------------
// End of network: jump here if step not active
// Jump to end of this FB if the step has been active to avoid
// execution of another step in the same scan
//---------------------------------
      JU    ENDS;
J29:  NOP   0;



NETWORK
TITLE = Step 420
// test first line without logic and rest with AND
// skip this network if stepnumber not equal to 420
      L     #stepnumber;
      L     420;
      ==I;
      JCN   J30;

//---------------------------------
// Actions (continuouss)
//---------------------------------

//---------------------------------
// --- TRANSITION TO S430 ---
//---------------------------------

// Transition Logic
      SET;  //make sure RLO is high so the transition can happen when no conditions present

      A     #XV003_OPN;  //XV003 opened
      A     #XV004_OPN;  //XV004 opened
      A     #XV005_OPN;  //XV005 opened
      JCN   L30;

      L     430;
      T     #stepnumber;

L30:  NOP   0;


D30:  NOP   0;

//---------------------------------
// End of network: jump here if step not active
// Jump to end of this FB if the step has been active to avoid
// execution of another step in the same scan
//---------------------------------
      JU    ENDS;
J30:  NOP   0;



NETWORK
TITLE = Step 430
// test first line without logic and rest with OR
// skip this network if stepnumber not equal to 430
      L     #stepnumber;
      L     430;
      ==I;
      JCN   J31;

//---------------------------------
// Actions (continuouss)
//---------------------------------

//---------------------------------
// --- TRANSITION TO S440 ---
//---------------------------------

// Transition Logic
      SET;  //make sure RLO is high so the transition can happen when no conditions present

      O     #XV003_OPN;  //XV003 opened
      O     #XV004_OPN;  //XV004 opened
      O     #XV005_OPN;  //XV005 opened
      JCN   L31;

      L     440;
      T     #stepnumber;

L31:  NOP   0;


D31:  NOP   0;

//---------------------------------
// End of network: jump here if step not active
// Jump to end of this FB if the step has been active to avoid
// execution of another step in the same scan
//---------------------------------
      JU    ENDS;
J31:  NOP   0;



NETWORK
TITLE = Step 440
// test button
// skip this network if stepnumber not equal to 440
      L     #stepnumber;
      L     440;
      ==I;
      JCN   J32;

//---------------------------------
// Actions (continuouss)
//---------------------------------

// Action: show button_1
      SET;
      =     #button_1_visible;

// Action: select text with ID 16: continue
      L     16;
      T     #button_1_text;

//---------------------------------
// --- TRANSITION TO S450 ---
//---------------------------------

// Transition Logic
      SET;  //make sure RLO is high so the transition can happen when no conditions present

      A     #button_1_pushed;  //button “continue”
      JCN   L32;

      L     450;
      T     #stepnumber;

L32:  NOP   0;


//---------------------------------
// Actions (last scan)
// This is immediately executed once the stepnumber changes
//---------------------------------
      L     #stepnumber;
      L     #previous_stepnumber;
      <>I;
      JCN   D32;

// Action: hide button_1
      CLR;
      =     #button_1_visible;


D32:  NOP   0;

//---------------------------------
// End of network: jump here if step not active
// Jump to end of this FB if the step has been active to avoid
// execution of another step in the same scan
//---------------------------------
      JU    ENDS;
J32:  NOP   0;



NETWORK
TITLE = Step 450
// test button with capital => no problem, the button is case insensitive
// skip this network if stepnumber not equal to 450
      L     #stepnumber;
      L     450;
      ==I;
      JCN   J33;

//---------------------------------
// Actions (continuouss)
//---------------------------------

// Action: show button_1
      SET;
      =     #button_1_visible;

// Action: select text with ID 17: ok
      L     17;
      T     #button_1_text;

//---------------------------------
// --- TRANSITION TO S460 ---
//---------------------------------

// Transition Logic
      SET;  //make sure RLO is high so the transition can happen when no conditions present

      A     #button_1_pushed;  //Button “ok”
      JCN   L33;

      L     460;
      T     #stepnumber;

L33:  NOP   0;


//---------------------------------
// Actions (last scan)
// This is immediately executed once the stepnumber changes
//---------------------------------
      L     #stepnumber;
      L     #previous_stepnumber;
      <>I;
      JCN   D33;

// Action: hide button_1
      CLR;
      =     #button_1_visible;


D33:  NOP   0;

//---------------------------------
// End of network: jump here if step not active
// Jump to end of this FB if the step has been active to avoid
// execution of another step in the same scan
//---------------------------------
      JU    ENDS;
J33:  NOP   0;



NETWORK
TITLE = Step 460
// test button without opening quotation marks => no problem, any marks are just removed
// skip this network if stepnumber not equal to 460
      L     #stepnumber;
      L     460;
      ==I;
      JCN   J34;

//---------------------------------
// Actions (continuouss)
//---------------------------------

// Action: show button_1
      SET;
      =     #button_1_visible;

// Action: select text with ID 18: cancel
      L     18;
      T     #button_1_text;

//---------------------------------
// --- TRANSITION TO S470 ---
//---------------------------------

// Transition Logic
      SET;  //make sure RLO is high so the transition can happen when no conditions present

      A     #button_1_pushed;  //button cancel”
      JCN   L34;

      L     470;
      T     #stepnumber;

L34:  NOP   0;


//---------------------------------
// Actions (last scan)
// This is immediately executed once the stepnumber changes
//---------------------------------
      L     #stepnumber;
      L     #previous_stepnumber;
      <>I;
      JCN   D34;

// Action: hide button_1
      CLR;
      =     #button_1_visible;


D34:  NOP   0;

//---------------------------------
// End of network: jump here if step not active
// Jump to end of this FB if the step has been active to avoid
// execution of another step in the same scan
//---------------------------------
      JU    ENDS;
J34:  NOP   0;



NETWORK
TITLE = Step 470
// test button without closing quotation marks => no problem, any marks are just removed
// skip this network if stepnumber not equal to 470
      L     #stepnumber;
      L     470;
      ==I;
      JCN   J35;

//---------------------------------
// Actions (continuouss)
//---------------------------------

// Action: show button_1
      SET;
      =     #button_1_visible;

// Action: select text with ID 19: go back
      L     19;
      T     #button_1_text;

//---------------------------------
// --- TRANSITION TO S480 ---
//---------------------------------

// Transition Logic
      SET;  //make sure RLO is high so the transition can happen when no conditions present

      A     #button_1_pushed;  //button “go back
      JCN   L35;

      L     480;
      T     #stepnumber;

L35:  NOP   0;


//---------------------------------
// Actions (last scan)
// This is immediately executed once the stepnumber changes
//---------------------------------
      L     #stepnumber;
      L     #previous_stepnumber;
      <>I;
      JCN   D35;

// Action: hide button_1
      CLR;
      =     #button_1_visible;


D35:  NOP   0;

//---------------------------------
// End of network: jump here if step not active
// Jump to end of this FB if the step has been active to avoid
// execution of another step in the same scan
//---------------------------------
      JU    ENDS;
J35:  NOP   0;



NETWORK
TITLE = Step 480
// test 3 buttons
// skip this network if stepnumber not equal to 480
      L     #stepnumber;
      L     480;
      ==I;
      JCN   J36;

//---------------------------------
// Actions (continuouss)
//---------------------------------

// Action: show button_1
      SET;
      =     #button_1_visible;

// Action: select text with ID 16: continue
      L     16;
      T     #button_1_text;

// Action: show button_2
      SET;
      =     #button_2_visible;

// Action: select text with ID 18: cancel
      L     18;
      T     #button_2_text;

// Action: show button_3
      SET;
      =     #button_3_visible;

// Action: select text with ID 19: go back
      L     19;
      T     #button_3_text;

//---------------------------------
// --- TRANSITION TO S490 ---
//---------------------------------

// Transition Logic
      SET;  //make sure RLO is high so the transition can happen when no conditions present

      A     #button_1_pushed;  //button “continue”
      A     #button_2_pushed;  //button “cancel”
      A     #button_3_pushed;  //button “go back”
      JCN   L36;

      L     490;
      T     #stepnumber;

L36:  NOP   0;


//---------------------------------
// Actions (last scan)
// This is immediately executed once the stepnumber changes
//---------------------------------
      L     #stepnumber;
      L     #previous_stepnumber;
      <>I;
      JCN   D36;

// Action: hide button_1
      CLR;
      =     #button_1_visible;

// Action: hide button_2
      CLR;
      =     #button_2_visible;

// Action: hide button_3
      CLR;
      =     #button_3_visible;


D36:  NOP   0;

//---------------------------------
// End of network: jump here if step not active
// Jump to end of this FB if the step has been active to avoid
// execution of another step in the same scan
//---------------------------------
      JU    ENDS;
J36:  NOP   0;



NETWORK
TITLE = Step 490
// test 4 buttons => not foreseen in the template, so should log an error
// skip this network if stepnumber not equal to 490
      L     #stepnumber;
      L     490;
      ==I;
      JCN   J37;

//---------------------------------
// Actions (continuouss)
//---------------------------------

// Action: show button_1
      SET;
      =     #button_1_visible;

// Action: select text with ID 16: continue
      L     16;
      T     #button_1_text;

// Action: show button_2
      SET;
      =     #button_2_visible;

// Action: select text with ID 18: cancel
      L     18;
      T     #button_2_text;

// Action: show button_3
      SET;
      =     #button_3_visible;

// Action: select text with ID 19: go back
      L     19;
      T     #button_3_text;

//---------------------------------
// --- TRANSITION TO S510 ---
//---------------------------------

// Transition Logic
      SET;  //make sure RLO is high so the transition can happen when no conditions present

      A     #button_1_pushed;  //button “continue”
      A     #button_2_pushed;  //button “cancel”
      A     #button_3_pushed;  //button “go back”
      JCN   L37;

      L     510;
      T     #stepnumber;

L37:  NOP   0;


//---------------------------------
// Actions (last scan)
// This is immediately executed once the stepnumber changes
//---------------------------------
      L     #stepnumber;
      L     #previous_stepnumber;
      <>I;
      JCN   D37;

// Action: hide button_1
      CLR;
      =     #button_1_visible;

// Action: hide button_2
      CLR;
      =     #button_2_visible;

// Action: hide button_3
      CLR;
      =     #button_3_visible;


D37:  NOP   0;

//---------------------------------
// End of network: jump here if step not active
// Jump to end of this FB if the step has been active to avoid
// execution of another step in the same scan
//---------------------------------
      JU    ENDS;
J37:  NOP   0;



NETWORK
TITLE = Step 510
// test message
// skip this network if stepnumber not equal to 510
      L     #stepnumber;
      L     510;
      ==I;
      JCN   J38;

//---------------------------------
// Actions (continuouss)
//---------------------------------

// Action: message “add the manual ingredients”
      L     21;
      T     #message;

//---------------------------------
// --- TRANSITION TO S520 ---
//---------------------------------

// Transition Logic
      SET;  //make sure RLO is high so the transition can happen when no conditions present

      JCN   L38;

      L     520;
      T     #stepnumber;

L38:  NOP   0;


//---------------------------------
// Actions (last scan)
// This is immediately executed once the stepnumber changes
//---------------------------------
      L     #stepnumber;
      L     #previous_stepnumber;
      <>I;
      JCN   D38;

// Action: clear message
      L     0;
      T     #message;


D38:  NOP   0;

//---------------------------------
// End of network: jump here if step not active
// Jump to end of this FB if the step has been active to avoid
// execution of another step in the same scan
//---------------------------------
      JU    ENDS;
J38:  NOP   0;



NETWORK
TITLE = Step 520
// test falseword with two words in transition
// skip this network if stepnumber not equal to 520
      L     #stepnumber;
      L     520;
      ==I;
      JCN   J39;

//---------------------------------
// Actions (continuouss)
//---------------------------------

//---------------------------------
// --- TRANSITION TO S530 ---
//---------------------------------

// Transition Logic
      SET;  //make sure RLO is high so the transition can happen when no conditions present

      AN    #XV003_OPN;  //XV003 not opened
      JCN   L39;

      L     530;
      T     #stepnumber;

L39:  NOP   0;


D39:  NOP   0;

//---------------------------------
// End of network: jump here if step not active
// Jump to end of this FB if the step has been active to avoid
// execution of another step in the same scan
//---------------------------------
      JU    ENDS;
J39:  NOP   0;



NETWORK
TITLE = Step 530
// test trueword with multiple words in action
// skip this network if stepnumber not equal to 530
      L     #stepnumber;
      L     530;
      ==I;
      JCN   J40;

//---------------------------------
// Actions (continuouss)
//---------------------------------

// Action: move to open position XV003
      SET;
      =     #XV003_CMD;

//---------------------------------
// --- TRANSITION TO S540 ---
//---------------------------------

// Transition Logic
      SET;  //make sure RLO is high so the transition can happen when no conditions present

      JCN   L40;

      L     540;
      T     #stepnumber;

L40:  NOP   0;


D40:  NOP   0;

//---------------------------------
// End of network: jump here if step not active
// Jump to end of this FB if the step has been active to avoid
// execution of another step in the same scan
//---------------------------------
      JU    ENDS;
J40:  NOP   0;



NETWORK
TITLE = Step 540
// test putting controller in auto with pulseword
// skip this network if stepnumber not equal to 540
      L     #stepnumber;
      L     540;
      ==I;
      JCN   J41;

//---------------------------------
// Actions (continuouss)
//---------------------------------

// Action: FIC001 auto
      SET;
      =     #FIC001_AUT;

//---------------------------------
// --- TRANSITION TO S550 ---
//---------------------------------

// Transition Logic
      SET;  //make sure RLO is high so the transition can happen when no conditions present

      JCN   L41;

      L     550;
      T     #stepnumber;

L41:  NOP   0;


D41:  NOP   0;

//---------------------------------
// End of network: jump here if step not active
// Jump to end of this FB if the step has been active to avoid
// execution of another step in the same scan
//---------------------------------
      JU    ENDS;
J41:  NOP   0;



NETWORK
TITLE = Step 550
// test putting controller in auto with pulseword consisting of multiple words
// skip this network if stepnumber not equal to 550
      L     #stepnumber;
      L     550;
      ==I;
      JCN   J42;

//---------------------------------
// Actions (continuouss)
//---------------------------------

// Action: FIC001 switch to auto
      SET;
      =     #FIC001_AUT;

//---------------------------------
// --- TRANSITION TO S560 ---
//---------------------------------

// Transition Logic
      SET;  //make sure RLO is high so the transition can happen when no conditions present

      JCN   L42;

      L     560;
      T     #stepnumber;

L42:  NOP   0;


D42:  NOP   0;

//---------------------------------
// End of network: jump here if step not active
// Jump to end of this FB if the step has been active to avoid
// execution of another step in the same scan
//---------------------------------
      JU    ENDS;
J42:  NOP   0;



NETWORK
TITLE = Step 560
// test with pulseword in front
// skip this network if stepnumber not equal to 560
      L     #stepnumber;
      L     560;
      ==I;
      JCN   J43;

//---------------------------------
// Actions (continuouss)
//---------------------------------

// Action: auto FIC001
      SET;
      =     #FIC001_AUT;

//---------------------------------
// --- TRANSITION TO S570 ---
//---------------------------------

// Transition Logic
      SET;  //make sure RLO is high so the transition can happen when no conditions present

      JCN   L43;

      L     570;
      T     #stepnumber;

L43:  NOP   0;


D43:  NOP   0;

//---------------------------------
// End of network: jump here if step not active
// Jump to end of this FB if the step has been active to avoid
// execution of another step in the same scan
//---------------------------------
      JU    ENDS;
J43:  NOP   0;



NETWORK
TITLE = Step 570
// test with pulseword in front
// skip this network if stepnumber not equal to 570
      L     #stepnumber;
      L     570;
      ==I;
      JCN   J44;

//---------------------------------
// Actions (continuouss)
//---------------------------------

// Action: switch to auto FIC001
      SET;
      =     #FIC001_AUT;

//---------------------------------
// --- TRANSITION TO S580 ---
//---------------------------------

// Transition Logic
      SET;  //make sure RLO is high so the transition can happen when no conditions present

      JCN   L44;

      L     580;
      T     #stepnumber;

L44:  NOP   0;


D44:  NOP   0;

//---------------------------------
// End of network: jump here if step not active
// Jump to end of this FB if the step has been active to avoid
// execution of another step in the same scan
//---------------------------------
      JU    ENDS;
J44:  NOP   0;



NETWORK
TITLE = Step 580
// test steptime in s
// skip this network if stepnumber not equal to 580
      L     #stepnumber;
      L     580;
      ==I;
      JCN   J45;

//---------------------------------
// Actions (continuouss)
//---------------------------------

//---------------------------------
// --- TRANSITION TO S590 ---
//---------------------------------

// Calculation:
      L     #steptime_s;
      L     2.0;
      >R;
      =     #B5;

// Transition Logic
      SET;  //make sure RLO is high so the transition can happen when no conditions present

      A     #B5;  //steptime > 2.0s
      JCN   L45;

      L     590;
      T     #stepnumber;

L45:  NOP   0;


D45:  NOP   0;

//---------------------------------
// End of network: jump here if step not active
// Jump to end of this FB if the step has been active to avoid
// execution of another step in the same scan
//---------------------------------
      JU    ENDS;
J45:  NOP   0;



NETWORK
TITLE = Step 590
// test steptime in m
// skip this network if stepnumber not equal to 590
      L     #stepnumber;
      L     590;
      ==I;
      JCN   J46;

//---------------------------------
// Actions (continuouss)
//---------------------------------

//---------------------------------
// --- TRANSITION TO S600 ---
//---------------------------------

// Calculation:
      L     #steptime_m;
      L     1.50;
      >R;
      =     #B6;

// Transition Logic
      SET;  //make sure RLO is high so the transition can happen when no conditions present

      A     #B6;  //steptime > 1.50m
      JCN   L46;

      L     600;
      T     #stepnumber;

L46:  NOP   0;


D46:  NOP   0;

//---------------------------------
// End of network: jump here if step not active
// Jump to end of this FB if the step has been active to avoid
// execution of another step in the same scan
//---------------------------------
      JU    ENDS;
J46:  NOP   0;



NETWORK
TITLE = Step 600
// test steptime in h
// skip this network if stepnumber not equal to 600
      L     #stepnumber;
      L     600;
      ==I;
      JCN   J47;

//---------------------------------
// Actions (continuouss)
//---------------------------------

//---------------------------------
// --- TRANSITION TO S610 ---
//---------------------------------

// Calculation:
      L     #steptime_h;
      L     4.3;
      >R;
      =     #B7;

// Transition Logic
      SET;  //make sure RLO is high so the transition can happen when no conditions present

      A     #B7;  //steptime > 4.3h
      JCN   L47;

      L     610;
      T     #stepnumber;

L47:  NOP   0;


D47:  NOP   0;

//---------------------------------
// End of network: jump here if step not active
// Jump to end of this FB if the step has been active to avoid
// execution of another step in the same scan
//---------------------------------
      JU    ENDS;
J47:  NOP   0;



NETWORK
TITLE = Step 610
// test steptime with unit separated by space => still works (because it takes the last character)
// skip this network if stepnumber not equal to 610
      L     #stepnumber;
      L     610;
      ==I;
      JCN   J48;

//---------------------------------
// Actions (continuouss)
//---------------------------------

//---------------------------------
// --- TRANSITION TO S640 ---
//---------------------------------

// Calculation:
      L     #steptime_m;
      L     1.50;
      >R;
      =     #B8;

// Transition Logic
      SET;  //make sure RLO is high so the transition can happen when no conditions present

      A     #B8;  //steptime > 1.50 m
      JCN   L48;

      L     640;
      T     #stepnumber;

L48:  NOP   0;


D48:  NOP   0;

//---------------------------------
// End of network: jump here if step not active
// Jump to end of this FB if the step has been active to avoid
// execution of another step in the same scan
//---------------------------------
      JU    ENDS;
J48:  NOP   0;



NETWORK
TITLE = Step 640
// test steptime with variable with unit
// skip this network if stepnumber not equal to 640
      L     #stepnumber;
      L     640;
      ==I;
      JCN   J49;

//---------------------------------
// Actions (continuouss)
//---------------------------------

//---------------------------------
// --- TRANSITION TO S650 ---
//---------------------------------

// Calculation:
      L     #steptime_h;
      L     #timesetting;
      >R;
      =     #B9;

// Transition Logic
      SET;  //make sure RLO is high so the transition can happen when no conditions present

      A     #B9;  //steptime > timesetting
      JCN   L49;

      L     650;
      T     #stepnumber;

L49:  NOP   0;


D49:  NOP   0;

//---------------------------------
// End of network: jump here if step not active
// Jump to end of this FB if the step has been active to avoid
// execution of another step in the same scan
//---------------------------------
      JU    ENDS;
J49:  NOP   0;



NETWORK
TITLE = Step 650
// reset a timer
// skip this network if stepnumber not equal to 650
      L     #stepnumber;
      L     650;
      ==I;
      JCN   J50;

//---------------------------------
// Actions (continuouss)
//---------------------------------

// Action: reset timer_dosing
      L     0.0;
      T     #timer_dosing_s;

//---------------------------------
// --- TRANSITION TO S660 ---
//---------------------------------

// Transition Logic
      SET;  //make sure RLO is high so the transition can happen when no conditions present

      JCN   L50;

      L     660;
      T     #stepnumber;

L50:  NOP   0;


D50:  NOP   0;

//---------------------------------
// End of network: jump here if step not active
// Jump to end of this FB if the step has been active to avoid
// execution of another step in the same scan
//---------------------------------
      JU    ENDS;
J50:  NOP   0;



NETWORK
TITLE = Step 660
// start a timer
// skip this network if stepnumber not equal to 660
      L     #stepnumber;
      L     660;
      ==I;
      JCN   J51;

//---------------------------------
// Actions (continuouss)
//---------------------------------

// Action: start timer_mixing
      CLR;
      =     #timer_mixing_pause;

//---------------------------------
// --- TRANSITION TO S670 ---
//---------------------------------

// Transition Logic
      SET;  //make sure RLO is high so the transition can happen when no conditions present

      JCN   L51;

      L     670;
      T     #stepnumber;

L51:  NOP   0;


D51:  NOP   0;

//---------------------------------
// End of network: jump here if step not active
// Jump to end of this FB if the step has been active to avoid
// execution of another step in the same scan
//---------------------------------
      JU    ENDS;
J51:  NOP   0;



NETWORK
TITLE = Step 670
// pause a timer
// skip this network if stepnumber not equal to 670
      L     #stepnumber;
      L     670;
      ==I;
      JCN   J52;

//---------------------------------
// Actions (continuouss)
//---------------------------------

// Action: pause timer_circulation
      SET;
      =     #timer_circulation_pause;

//---------------------------------
// --- TRANSITION TO S680 ---
//---------------------------------

// Transition Logic
      SET;  //make sure RLO is high so the transition can happen when no conditions present

      JCN   L52;

      L     680;
      T     #stepnumber;

L52:  NOP   0;


D52:  NOP   0;

//---------------------------------
// End of network: jump here if step not active
// Jump to end of this FB if the step has been active to avoid
// execution of another step in the same scan
//---------------------------------
      JU    ENDS;
J52:  NOP   0;



NETWORK
TITLE = Step 680
// test timer in m
// skip this network if stepnumber not equal to 680
      L     #stepnumber;
      L     680;
      ==I;
      JCN   J53;

//---------------------------------
// Actions (continuouss)
//---------------------------------

//---------------------------------
// --- TRANSITION TO S690 ---
//---------------------------------

// Calculation:
      L     #timer_dosing_m;
      L     5.2;
      >=R;
      =     #B10;

// Transition Logic
      SET;  //make sure RLO is high so the transition can happen when no conditions present

      A     #B10;  //timer_dosing >= 5.2 m
      JCN   L53;

      L     690;
      T     #stepnumber;

L53:  NOP   0;


D53:  NOP   0;

//---------------------------------
// End of network: jump here if step not active
// Jump to end of this FB if the step has been active to avoid
// execution of another step in the same scan
//---------------------------------
      JU    ENDS;
J53:  NOP   0;



NETWORK
TITLE = Step 690
// test timer with variable with unit
// skip this network if stepnumber not equal to 690
      L     #stepnumber;
      L     690;
      ==I;
      JCN   J54;

//---------------------------------
// Actions (continuouss)
//---------------------------------

//---------------------------------
// --- TRANSITION TO S700 ---
//---------------------------------

// Calculation:
      L     #timer_circulation_h;
      L     #timesetting;
      <R;
      =     #B11;

// Transition Logic
      SET;  //make sure RLO is high so the transition can happen when no conditions present

      A     #B11;  //timer_circulation < timesetting
      JCN   L54;

      L     700;
      T     #stepnumber;

L54:  NOP   0;


D54:  NOP   0;

//---------------------------------
// End of network: jump here if step not active
// Jump to end of this FB if the step has been active to avoid
// execution of another step in the same scan
//---------------------------------
      JU    ENDS;
J54:  NOP   0;



NETWORK
TITLE = Step 700
// test putting a controller in manual
// skip this network if stepnumber not equal to 700
      L     #stepnumber;
      L     700;
      ==I;
      JCN   J55;

//---------------------------------
// Actions (continuouss)
//---------------------------------

// Action: FIC001 manual
      CLR;
      =     #FIC001_AUT;

//---------------------------------
// --- TRANSITION TO S710 ---
//---------------------------------

// Transition Logic
      SET;  //make sure RLO is high so the transition can happen when no conditions present

      JCN   L55;

      L     710;
      T     #stepnumber;

L55:  NOP   0;


D55:  NOP   0;

//---------------------------------
// End of network: jump here if step not active
// Jump to end of this FB if the step has been active to avoid
// execution of another step in the same scan
//---------------------------------
      JU    ENDS;
J55:  NOP   0;



NETWORK
TITLE = Step 710
// test putting a controller in manual while changing the output value
// skip this network if stepnumber not equal to 710
      L     #stepnumber;
      L     710;
      ==I;
      JCN   J56;

//---------------------------------
// Actions (first scan)
//---------------------------------
      A     #initial_scan;
      JCN   C56;

// Action: FIC001_VAL_OUT = 20.0
      L     20.0;
      T     #FIC001_VAL_OUT;

// Action: FIC001_SET_OUT = true
      SET;
      =     #FIC001_SET_OUT;

      JU    D56;
C56:  NOP   0;


//---------------------------------
// Actions (continuouss)
//---------------------------------

// Action: FIC001 manual 20.0
      CLR;
      =     #FIC001_AUT;

// Action: FIC001_SET_OUT = false
      CLR;
      =     #FIC001_SET_OUT;

//---------------------------------
// --- TRANSITION TO S720 ---
//---------------------------------

// Transition Logic
      SET;  //make sure RLO is high so the transition can happen when no conditions present

      JCN   L56;

      L     720;
      T     #stepnumber;

L56:  NOP   0;

